TYPE ST_PMLControl :
STRUCT
	bNewCommand		: BOOL;
	bConfirmation	: BOOL;
	
	eMode			: E_PMLUnitMode;
	eModeCommand	: E_PMLUnitMode;
	
	eState			: E_PMLState;
	eStateCommand	: E_PMLCommand;
	
	a_sModeNames	: ARRAY[0..31] OF STRING;
END_STRUCT
END_TYPE

(* stored: Version 1.1.0.1, ProductVersion 3.1.4024.9
   DUT ST_PMLControl: Id {b98df5eb-74fe-4f0b-aa48-e46153fa07dc} *)
